PROGRAM MAIN
VAR
  	(* JSON document *)
	fbJson 			: FB_JsonSaxReader;
	pJsonParse		: JsonSaxHandler;
	sJsonDoc 		: STRING(255) := '{"Values":{"Timestamp":"2017-04-04T12:42:42","Sensor1":42.42,"Sensor2":42}}';	
END_VAR

fbJson.Parse(sJson := sJsonDoc, ipHdl := pJsonParse);

END_PROGRAM

(* stored: Version 1.1.0.1, ProductVersion 3.1.4021.12
   POU MAIN: Id {b49b0a40-e0b7-411b-a0ef-9b7ce6587010}, SpecialFunc None *)
